Yaskawa INFORM job: LESLE2.JBI

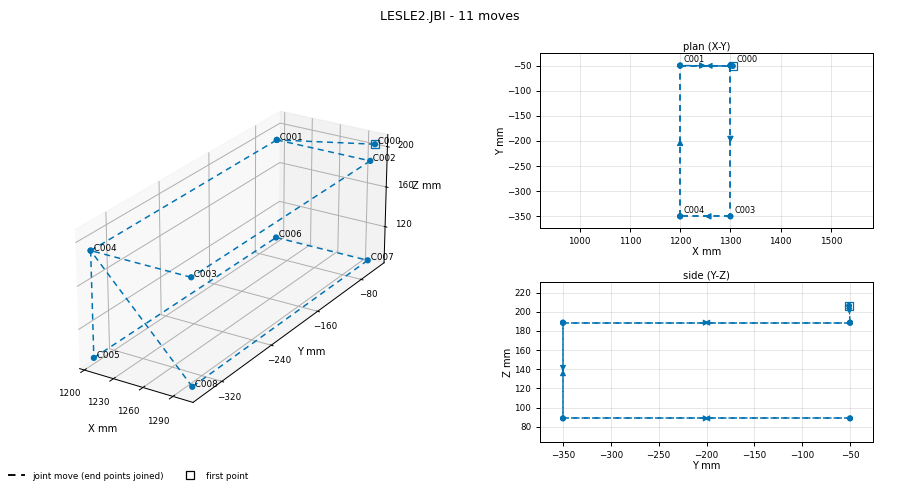
[picture p0: tool path of LESLE2.JBI, 11 of 11 moves have a stored position in this frame; points joined in program order, loops and branches not executed]
/JOB
//NAME LESLE2
//POS
///NPOS 11,0,0,0
///TOOL 0
///RECTAN
///RCONF 0,0,0,0,0
C000=1304.952,-51.025,206.350,-168.80,-11.35,-67.97
C001=1200.000,-50.000,188.655,-168.81,-11.35,-67.96
C002=1300.000,-50.000,188.655,-168.80,-11.35,-67.96
C003=1300.000,-350.000,188.655,-168.80,-11.35,-67.96
C004=1200.000,-350.000,188.655,-168.80,-11.35,-67.94
C005=1200.000,-350.000,88.655,-168.78,-11.34,-67.97
C006=1200.000,-50.000,88.655,-168.79,-11.36,-67.95
C007=1300.000,-50.000,88.655,-168.76,-11.35,-67.97
C008=1300.000,-350.000,88.655,-168.75,-11.34,-67.99
C009=1200.000,-350.000,188.655,-168.75,-11.34,-67.98
C010=1200.000,-50.000,188.655,-168.75,-11.33,-67.99
//INST
///DATE 2014/11/02 00:23
///ATTR 0,0,0,0,0,0,0,0,0,0,0,0,1,1,0,0
///FRAME BASE
NOP
*1
MOVJ C000 VJ=25.00 CONT
MOVJ C001 VJ=25.00 CONT
MOVJ C002 VJ=25.00 CONT
MOVJ C003 VJ=25.00 CONT
MOVJ C004 VJ=25.00 CONT
MOVJ C005 VJ=25.00 CONT
MOVJ C006 VJ=25.00 CONT
MOVJ C007 VJ=25.00 CONT
MOVJ C008 VJ=25.00 CONT
MOVJ C009 VJ=25.00 CONT
MOVJ C010 VJ=25.00 CONT
JUMP *1
END
